Staubli VAL3: onStart.pgx

program onStart()
  local num i
  local num l_nIndex
  local bool l_bOk
begin
  cls()
  // reset the Key pressure
  call use:nullKey(nKey)
  setTextMode(0)
  // build the list
  call buildList()
  nRefresh=clock()
 call refreshStatic()
end
